// TwinCAT 3 PLC project TwinCAT_NC_Sample_PTP_Move
// libraries:
//   Tc2_Math, * (Beckhoff Automation GmbH)
//   Tc2_MC2, * (Beckhoff Automation GmbH)
//   Tc2_Standard, * (Beckhoff Automation GmbH)
//   Tc2_System, * (Beckhoff Automation GmbH)
//   Tc3_Module, * (Beckhoff Automation GmbH)
// project tree:
//   Data types/ MoveState_t.TcDUT
//   Global Variables/ Globale_Variablen.TcGVL, TwinCAT_Configuration.TcGVL, Variablen_Konfiguration.TcGVL
//   POUs/ MAIN.TcPOU
//   / Standard.TcTTO
// real-time tasks:
//   TASK Standard: cycle T#10ms, priority 20, ADS port 350
// motion (NC):
//   TASK NC-Task 1 SAF: cycle T#2ms, priority 4, ADS port 501
//   TASK NC-Task 1 SVB: cycle T#10ms, priority 8, ADS port 511
//   AXIS Axis 1 (id 1)
//     Dynamic: AccelerationMaximum=10000, DecelerationMaximum=10000
//     Velo: FastManual=300
//     MotionControl: Range=5, Time=0.1
//     encoder EncType=1
//       EncPara: ScaleFactorNumerator=90, ScaleFactorDenominator=65535
//         Sim: RandScale=0.1
//     drive DrvType=5
//       Analog: SmoothingFilterOrder=0, SmoothingFilterTime=0
//       TimeComp: DriveDelayCycles=0, TaskDelayCycles=1
//     controller CtrType=3
//       CtrPara: PriorControlFactor=1
//         Observer: BandWidth=20
// I/O:
//   DEVICE Device 1 (EtherCAT) (disabled), AmsNetId 192.168.2.43.2.1
//     Drive 1 (CMMP-AS V4p0 CiA402) [CMMP-AS V4p0 CiA402]
// variable links:
//   TwinCAT_NC_Sample_PTP_Move/TwinCAT_NC_Sample_PTP_Move Instance <-> NC-Task 1 SAF/Axes/Axis 1
//     Standard Inputs/MAIN.Axis1.NcToPlc <-> Outputs/Axis 1_ToPlc
//     Standard Outputs/MAIN.Axis1.PlcToNc <-> Inputs/Axis 1_FromPlc

CONFIGURATION TwinCAT_NC_Sample_PTP_Move
    RESOURCE PLC ON TwinCAT3
        TASK Standard(INTERVAL := T#10ms, PRIORITY := 20);
        PROGRAM MAIN WITH Standard : MAIN;
    END_RESOURCE
END_CONFIGURATION

// ---- Data types/MoveState_t.TcDUT
TYPE MoveState_t :
(
	MOVESTATE_INIT,
	MOVESTATE_ENABLE,
	MOVESTATE_FORWARD,
	MOVESTATE_BACKWARDS,
	MOVESTATE_BACKWARDSSLOW,
	MOVESTATE_NEWTARGETPOSITION,
	MOVESTATE_ERROR,
	MOVESTATE_RESET
);
END_TYPE

// ---- Global Variables/Globale_Variablen.TcGVL
{attribute 'Tc2GvlVarNames'}
VAR_GLOBAL
END_VAR

// ---- Global Variables/TwinCAT_Configuration.TcGVL
{attribute 'Tc2GvlVarNames'}
(* Generated automatically by TwinCAT - (read only) *)
VAR_CONFIG
	MAIN.Axis1.PlcToNc AT %QB0 : PLCTONC_AXIS_REF;
	MAIN.Axis1.NcToPlc AT %IB0 : NCTOPLC_AXIS_REF;
END_VAR

// ---- Global Variables/Variablen_Konfiguration.TcGVL
{attribute 'Tc2GvlVarNames'}
VAR_CONFIG
END_VAR

// ---- POUs/MAIN.TcPOU
PROGRAM MAIN
VAR
	Axis1 : AXIS_REF;					(* axis reference data structure *)
	state: MoveState_t;				(* state machine state *)

	PowerAxis1: MC_Power;
	PowerAxis1Out: ST_McOutputs;		(* debug function block output data *)

	MoveAxis1: MC_MoveAbsolute;
	MoveAbsoluteOut1: ST_McOutputs;	(* debug function block output data *)

	MoveAxis2: MC_MoveAbsolute;
	MoveAbsoluteOut2: ST_McOutputs;	(* debug function block output data *)

	Reset: MC_Reset;
	ResetOut : ST_McOutputs;			(* debug function block output data *)
END_VAR

	(* update the axis status at the beginning of each cycle *)
		Axis1.ReadStatus();

	(* move axis using a state machine *)
	CASE state OF

		MOVESTATE_INIT :	(* initialisation *)
			(* initialize all function blocks *)
			MoveAxis1.Execute := FALSE;
			MoveAxis2.Execute := FALSE;
			Reset.Execute := FALSE;
			state := MOVESTATE_ENABLE;

		MOVESTATE_ENABLE :
			PowerAxis1.Enable := TRUE;
			PowerAxis1.Enable_Positive := TRUE;
			PowerAxis1.Enable_Negative := TRUE;
			IF PowerAxis1.Status THEN
				state := MOVESTATE_FORWARD;
			ELSIF PowerAxis1.Error THEN
				state := MOVESTATE_ERROR;
			END_IF

		MOVESTATE_FORWARD :		(* start to first position *)
			MoveAxis1.Position := 1500;		(* start to intermediate tartet position *)
			MoveAxis1.Velocity := 500;		(* medium velocity level *)
			MoveAxis1.BufferMode := MC_Buffered;
			MoveAxis1.Execute := TRUE;
			IF MoveAxis1.Active  THEN
				(* axis is executing job but is not yet finished *)
				MoveAxis1.Execute := FALSE;
				(* leave this state and buffer a second command *)
				state := MOVESTATE_NEWTARGETPOSITION;
			ELSIF MoveAxis1.CommandAborted OR MoveAxis1.Error THEN
				state := MOVESTATE_ERROR;
			END_IF

		MOVESTATE_NEWTARGETPOSITION :		(* change target position while moving *)
			(* start a buffered motion command while axis is moving *)
			MoveAxis2.Position := 5000;		(* start to final target *)
			MoveAxis2.Velocity := 1500;		(* increase velocity *)
			MoveAxis2.BufferMode := MC_BlendingPrevious; 	(* use velocity of previous command till intermediate target position position *)
			MoveAxis2.Execute := TRUE;
			IF MoveAxis2.Done THEN
				MoveAxis2.Execute := FALSE;
				state := MOVESTATE_BACKWARDS;
			ELSIF MoveAxis2.CommandAborted OR MoveAxis2.Error THEN
				state := MOVESTATE_ERROR;
			END_IF

		MOVESTATE_BACKWARDS :	(* move back to initial position *)
			MoveAxis1.Position := 100;		(* position close to initial position *)
			MoveAxis1.Velocity := 2000;		(* high velocity *)
			MoveAxis1.BufferMode := MC_Buffered;
			MoveAxis1.Execute := TRUE;
			IF MoveAxis1.Active THEN
				(* axis is executing job but is not yet finished *)
				MoveAxis1.Execute := FALSE;
				(* leave this state and buffer a second command *)
				state := MOVESTATE_BACKWARDSSLOW;
			ELSIF MoveAxis1.CommandAborted OR MoveAxis1.Error THEN
				state := MOVESTATE_ERROR;
			END_IF

		MOVESTATE_BACKWARDSSLOW :	(* move back to initial position *)
			(* start a buffered motion command while axis is moving *)
			MoveAxis2.Position := 0;	(* back to initial position *)
			MoveAxis2.Velocity := 100; 	(* slow velocity *)
			MoveAxis2.BufferMode := MC_BlendingNext; 	(* use velocity from first target position *)
			MoveAxis2.Execute := TRUE;
			IF MoveAxis2.Done THEN
				MoveAxis2.Execute := FALSE;
				state := MOVESTATE_FORWARD;
			ELSIF MoveAxis2.CommandAborted OR MoveAxis2.Error THEN
				state := MOVESTATE_ERROR;
			END_IF

		MOVESTATE_ERROR :
			IF Axis1.Status.Error THEN
				state := MOVESTATE_RESET;	(* axis error requires reset *)
			ELSE
				state := MOVESTATE_INIT;		(* function block errors don't need a reset *)
			END_IF

		MOVESTATE_RESET :
			Reset.Execute := TRUE;
			IF Reset.Done THEN
				state := MOVESTATE_INIT;
			ELSIF Reset.Error THEN
				state := MOVESTATE_INIT; (* can't do anything here *)
			END_IF

	END_CASE

		ActPower();	(* call the power function block *)
		ActMove();	(* call the move function block *)
		ActReset();	(* call the reset function block *)

ACTION ActMove:
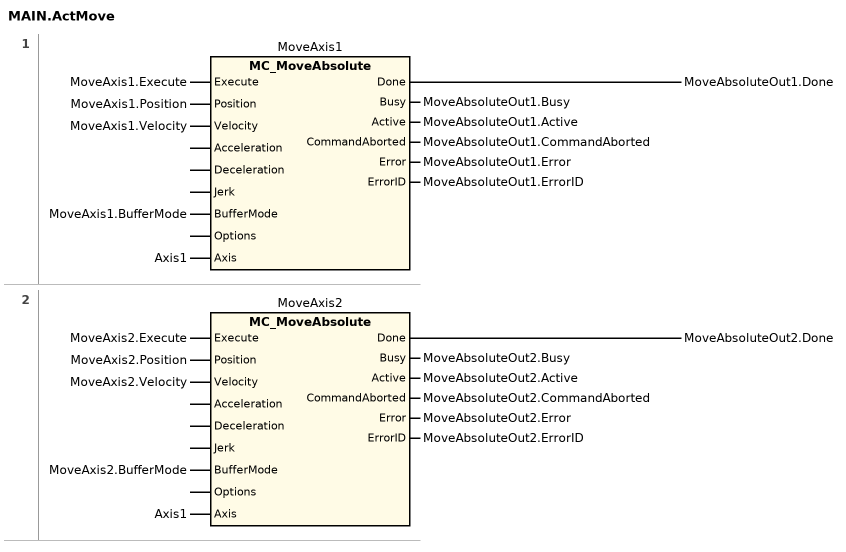
// NETWORK 1
MoveAxis1(
    Execute := MoveAxis1.Execute,
    Position := MoveAxis1.Position,
    Velocity := MoveAxis1.Velocity,
    BufferMode := MoveAxis1.BufferMode,
    Axis := Axis1,
    Busy => MoveAbsoluteOut1.Busy,
    Active => MoveAbsoluteOut1.Active,
    CommandAborted => MoveAbsoluteOut1.CommandAborted,
    Error => MoveAbsoluteOut1.Error,
    ErrorID => MoveAbsoluteOut1.ErrorID); // MC_MoveAbsolute
MoveAbsoluteOut1.Done := MoveAxis1.Done;

// NETWORK 2
MoveAxis2(
    Execute := MoveAxis2.Execute,
    Position := MoveAxis2.Position,
    Velocity := MoveAxis2.Velocity,
    BufferMode := MoveAxis2.BufferMode,
    Axis := Axis1,
    Busy => MoveAbsoluteOut2.Busy,
    Active => MoveAbsoluteOut2.Active,
    CommandAborted => MoveAbsoluteOut2.CommandAborted,
    Error => MoveAbsoluteOut2.Error,
    ErrorID => MoveAbsoluteOut2.ErrorID); // MC_MoveAbsolute
MoveAbsoluteOut2.Done := MoveAxis2.Done;
END_ACTION

ACTION ActPower:
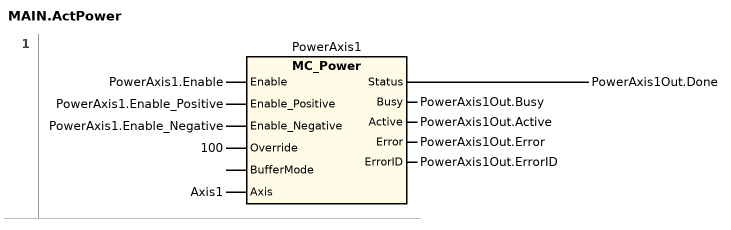
// NETWORK 1
PowerAxis1(
    Enable := PowerAxis1.Enable,
    Enable_Positive := PowerAxis1.Enable_Positive,
    Enable_Negative := PowerAxis1.Enable_Negative,
    Override := 100,
    Axis := Axis1,
    Busy => PowerAxis1Out.Busy,
    Active => PowerAxis1Out.Active,
    Error => PowerAxis1Out.Error,
    ErrorID => PowerAxis1Out.ErrorID); // MC_Power
PowerAxis1Out.Done := PowerAxis1.Status;
END_ACTION

ACTION ActReset:
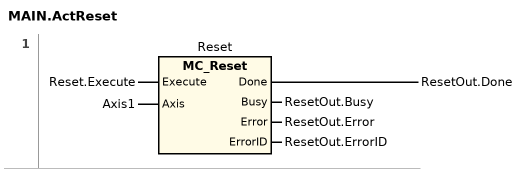
// NETWORK 1
Reset(
    Execute := Reset.Execute,
    Axis := Axis1,
    Busy => ResetOut.Busy,
    Error => ResetOut.Error,
    ErrorID => ResetOut.ErrorID); // MC_Reset
ResetOut.Done := Reset.Done;
END_ACTION

END_PROGRAM
